// TIA Portal V17 export
// export: Created 2022-07-20T07:01:30.4433567Z, ExportSetting WithDefaults, DisplayName Totally Integrated Automation Portal, DisplayVersion V17, DisplayName TIA Portal Openness, DisplayVersion V17, DisplayName TIA Portal Version Control Interface, DisplayVersion V17, DisplayName SINAMICS Startdrive Advanced, DisplayVersion V17, DisplayName SINAMICS Startdrive G130, G150, S120, S150, SINAMICS MV, S210, DisplayVersion V17, DisplayName SINAMICS Startdrive G110M, G120, G120C, G120D, G120P, G115D, DisplayVersion V17, DisplayName STEP 7 Professional, DisplayVersion V17, DisplayName STEP 7 Safety, DisplayVersion V17, DisplayName WinCC Advanced, DisplayVersion V17
FUNCTION_BLOCK "FB10281_3BeltsSystem_Control"   // FB10281, LAD
{ S7_Optimized_Access := 'TRUE' }
VERSION : 0.1
// stored: AutoNumber false, IsIECCheckEnabled false, IsRetainMemResEnabled false, MemoryReserve 100, SetENOAutomatically false, UDAEnableTagReadback false
   VAR_INPUT
      "3BeltsSystemCommunicationIn" : "st3BeltsSystemControlCommunicationIn";
      OmacState : Int;
      PresetCounter : UDInt;
   END_VAR
   VAR_OUTPUT
      "3BeltsSystemCommunicationOut" : "st3BeltsSystemControlCommunicationOut";
      HomingMode : Bool;
      AutomationMode : Bool;
      MotorsHomingDone : Bool;
      "3BeltsSystemReady" : Bool;
      AllFansRunning : Bool;
      EmptyRunOringActive : Bool;
      EmptyRunActive : Bool;
      PresetActualCounter : UDInt;
      ErrorBottomConveyor : Bool;
      ErrorUpperConveyor : Bool;
      ErrorFeederStacker : Bool;
   END_VAR
   VAR_IN_OUT
      RequestInitialization : Bool;
      RequestOperationModeHoming : Bool;
      RequestOperationModeAutomatic : Bool;
      RequestStart : Bool;
      RequestEmptyRun : Bool;
      RequestEmptyRunOring : Bool;
      RequestEmptyRunDone : Bool;
      RequestResetPressetCounter : Bool;
      RequestResetJobCounter : Bool;
      RequestStopFeeder : Bool;
      RequestFansOn : Bool;
      RequestFansOff : Bool;
      RequestNormalStop : Bool;
      RequestQuickStop : Bool;
      RequestEmergencyStop : Bool;
      RequestAcknowledge : Bool;
   END_VAR
   VAR
      RequestOperationModeHoming_Pulse : Bool;
      RequestOperationModeAutomatic_Pulse : Bool;
      RequestInitialization_Pulse : Bool;
      RequestFansOn_Pulse : Bool;
      RequestFansOff_Pulse : Bool;
      RequestStart_Pulse : Bool;
      RequestNormalStop_Pulse : Bool;
      R_TRIG_RequestInitialization : R_TRIG;
      R_TRIG_MotorsHomingDone { S7_SetPoint := 'True'} : R_TRIG;
      R_TRIG_RequestEmergencyStop { S7_SetPoint := 'True'} : R_TRIG;
      R_TRIG_RequestAcknowledge { S7_SetPoint := 'True'} : R_TRIG;
      R_TRIG_ResetPB { S7_SetPoint := 'True'} : R_TRIG;
      F_TRIG_In_3BeltsSystemReady { S7_SetPoint := 'True'} : F_TRIG;
      F_TRIG_ResetButton { S7_SetPoint := 'True'} : F_TRIG;
      TON_RequestInitialization { S7_SetPoint := 'True'} : TON_TIME;
      TON_MotorsHomingDone { S7_SetPoint := 'True'} : TON_TIME;
      TON_RequestEmergencyStop { S7_SetPoint := 'True'} : TON_TIME;
      TON_RequestAcknowledge { S7_SetPoint := 'True'} : TON_TIME;
      TON_AllFansRunning { S7_SetPoint := 'True'} : TON_TIME;
      FB10003_RequestOperationModeHoming_Pulse { S7_SetPoint := 'True'} : "FB10003_Pulse";
      FB10003_RequestOperationModeAutomatic_Pulse { S7_SetPoint := 'True'} : "FB10003_Pulse";
      FB10003_RequestInitialization_Pulse { S7_SetPoint := 'True'} : "FB10003_Pulse";
      FB10003_RequestStart_Pulse { S7_SetPoint := 'True'} : "FB10003_Pulse";
      FB10003_RequestNormalStop_Pulse { S7_SetPoint := 'True'} : "FB10003_Pulse";
      FB10003_RequestFansOn_Pulse { S7_SetPoint := 'True'} : "FB10003_Pulse";
      FB10003_RequestFansOff_Pulse { S7_SetPoint := 'True'} : "FB10003_Pulse";
   END_VAR
   VAR_TEMP
      na : Byte;
   END_VAR
BEGIN

REGION Network 1 (SCL): First Scan
   IF "FirstScan" THEN
       #"3BeltsSystemCommunicationOut".RequestInitialization := FALSE;
       #"3BeltsSystemCommunicationOut".DoStart := FALSE;
       #"3BeltsSystemCommunicationOut".DoNormalStop := FALSE;
       #"3BeltsSystemCommunicationOut".DoQuickStop := FALSE;
       #"3BeltsSystemCommunicationOut".DoEmergencyStop := FALSE;
       #"3BeltsSystemCommunicationOut".DoAcknowledge := FALSE;
       #"3BeltsSystemCommunicationOut".DoEmptyRun := FALSE;
       #"3BeltsSystemReady" := FALSE;
   END_IF;
END_REGION

REGION Network 2 (SCL): Edge Signals, Timers & Pulses
   REGION EDGE SIGNALS
       #R_TRIG_RequestInitialization(CLK := #RequestInitialization);
       #R_TRIG_RequestEmergencyStop(CLK := #RequestEmergencyStop);
       #R_TRIG_RequestAcknowledge(CLK := #RequestAcknowledge);
       #R_TRIG_ResetPB(CLK := #"3BeltsSystemCommunicationIn".ResetPB);
       #R_TRIG_MotorsHomingDone(CLK := #"3BeltsSystemCommunicationIn".MotorsHomingDone);

       #F_TRIG_In_3BeltsSystemReady(CLK := #"3BeltsSystemCommunicationIn"."3BeltsSystemReady");
       #F_TRIG_ResetButton(CLK := #"3BeltsSystemCommunicationIn".ResetPB);
   END_REGION

   REGION TIMERS
       #TON_RequestInitialization(IN := #RequestInitialization AND #"3BeltsSystemCommunicationOut".RequestInitialization,
                                  PT := T#1s);
       #TON_MotorsHomingDone(IN := #MotorsHomingDone,
                             PT := T#10s);
       #TON_RequestEmergencyStop(IN := #RequestEmergencyStop AND #"3BeltsSystemCommunicationOut".DoEmergencyStop,
                                 PT := T#1s);
       #TON_RequestAcknowledge(IN := #RequestAcknowledge AND #"3BeltsSystemCommunicationOut".DoAcknowledge,
                               PT := T#1s);
       #TON_AllFansRunning(IN := #"3BeltsSystemCommunicationIn".FansRunning,
                           PT := T#15s);
   END_REGION

   REGION PULSE
       #FB10003_RequestOperationModeHoming_Pulse(CLK := #RequestOperationModeHoming,
                                                 PT := T#200ms,
                                                 Q := #RequestOperationModeHoming_Pulse);
       #FB10003_RequestOperationModeAutomatic_Pulse(CLK := #RequestOperationModeAutomatic,
                                                    PT := T#200ms,
                                                    Q := #RequestOperationModeAutomatic_Pulse);
       #FB10003_RequestInitialization_Pulse(CLK := #RequestInitialization,
                                            PT := T#200ms,
                                            Q := #RequestInitialization_Pulse);
       #FB10003_RequestStart_Pulse(CLK := #RequestStart,
                                   PT := T#200ms,
                                   Q := #RequestStart_Pulse);
       #FB10003_RequestNormalStop_Pulse(CLK := #RequestNormalStop,
                                        PT := T#200ms,
                                        Q := #RequestNormalStop_Pulse);
       #FB10003_RequestFansOn_Pulse(CLK := #RequestFansOn,
                                    PT := T#100ms,
                                    Q := #RequestFansOn_Pulse);

       #FB10003_RequestFansOff_Pulse(CLK := #RequestFansOff,
                                     PT := T#100ms,
                                     Q := #RequestFansOff_Pulse);
   END_REGION
END_REGION

REGION Network 3 (SCL): 3BeltsSystems Commands Management
   #"3BeltsSystemCommunicationOut".RequestInitialization := #RequestInitialization;
   #"3BeltsSystemCommunicationOut".DoStart := #RequestStart_Pulse;
   #"3BeltsSystemCommunicationOut".DoNormalStop := #RequestNormalStop_Pulse;
   #"3BeltsSystemCommunicationOut".DoQuickStop := #RequestQuickStop;
   #"3BeltsSystemCommunicationOut".DoEmergencyStop := #RequestEmergencyStop;
   #"3BeltsSystemCommunicationOut".DoAcknowledge := #RequestAcknowledge;
   #"3BeltsSystemCommunicationOut".ResetPresetCounter := #RequestResetPressetCounter;
   #"3BeltsSystemCommunicationOut".RequestStopFeeder := #RequestStopFeeder;
   #"3BeltsSystemCommunicationOut".RequestFansOn := #RequestFansOn;
   #"3BeltsSystemCommunicationOut".RequestFansOff := #RequestFansOff;
   #"3BeltsSystemCommunicationOut".DoEmptyRun := #RequestEmptyRun;
   #"3BeltsSystemCommunicationOut".DoEmptyRunOring := #RequestEmptyRunOring;
   #"3BeltsSystemCommunicationOut".EmptyRunDone := #RequestEmptyRunDone;
   #"3BeltsSystemCommunicationOut".MachineInProduction := (#OmacState >= "OMAC_STATE_RESETTING") AND (#OmacState <= "OMAC_STATE_COMPLETE");
   #"3BeltsSystemCommunicationOut".ResetJobCounter := #RequestResetJobCounter;
   #"3BeltsSystemCommunicationOut".RequestInitialization := #RequestInitialization_Pulse;
   #"3BeltsSystemCommunicationOut".RequestOperationModeAutomatic := #RequestOperationModeAutomatic_Pulse;
   #"3BeltsSystemCommunicationOut".RequestOperationModeHoming := #RequestOperationModeHoming_Pulse;

   "FC10331_UDintTo4Bytes"(UDint := #PresetCounter,
                           Byte_0 => #"3BeltsSystemCommunicationOut".SetPresetCounterLowByte,
                           Byte_1 => #"3BeltsSystemCommunicationOut".SetPresetCounterHighByte,
                           Byte_2 => #na,
                           Byte_3 => #na);


   IF #R_TRIG_ResetPB.Q THEN
       #RequestAcknowledge := TRUE;
   ELSIF #F_TRIG_ResetButton.Q THEN
       #RequestAcknowledge := FALSE;
   END_IF;
END_REGION

REGION Network 4 (SCL): 3BeltsSystems States Management
   #"3BeltsSystemReady" := #"3BeltsSystemCommunicationIn"."3BeltsSystemReady";
   #HomingMode := #"3BeltsSystemCommunicationIn".HomingMode;
   #AutomationMode := #"3BeltsSystemCommunicationIn".AutomationMode;
   #ErrorUpperConveyor := #"3BeltsSystemCommunicationIn".ErrorUpperConveyor;
   #ErrorBottomConveyor := #"3BeltsSystemCommunicationIn".ErrorBottomConveyor;
   #ErrorFeederStacker := #"3BeltsSystemCommunicationIn".ErrorFeederStacker;
   #EmptyRunActive := #"3BeltsSystemCommunicationIn".EmptyRunActive;
   #EmptyRunOringActive := #"3BeltsSystemCommunicationIn".EmptyRunOringActive;
   #PresetActualCounter := "FC10330_2BytesToUDint"(LowByte := #"3BeltsSystemCommunicationIn".PresetActualCounterLowByte, HighByte := #"3BeltsSystemCommunicationIn".PresetActualCounterHighByte);
   IF #TON_AllFansRunning.Q THEN
       #AllFansRunning := TRUE;
   ELSE
       #AllFansRunning := FALSE;
   END_IF;
   IF #R_TRIG_MotorsHomingDone.Q THEN
       #MotorsHomingDone := TRUE;
   ELSIF #TON_MotorsHomingDone.Q THEN
       #MotorsHomingDone := FALSE;
   END_IF;
END_REGION
END_FUNCTION_BLOCK
